FUNCTION_BLOCK FB_SaMElementUndefined EXTENDS FB_SaMElement
VAR
END_VAR

METHOD FB_init : BOOL
VAR_INPUT
	bInitRetains : BOOL; // if TRUE, the retain variables are initialized (warm start / cold start)
	bInCopyCode : BOOL;  // if TRUE, the instance afterwards gets moved into the copy code (online change)
END_VAR
THIS^.SetText (eLocation := E_BaseLocation.pl, wsDescription := "Nieokreślony");
THIS^.SetText (eLocation := E_BaseLocation.en, wsDescription := "Undefined");
THIS^.SetText (eLocation := E_BaseLocation.de, wsDescription := "Nicht definiert");
THIS^.SetName (stName := THIS^.GetTexts ());
END_METHOD

END_FUNCTION_BLOCK

(* stored: Version 1.1.0.1
   POU FB_SaMElementUndefined: Id {57cb239a-4f66-0563-155d-52bfe19a13e5}, SpecialFunc None
   Method FB_init: Id {8424b7bd-9912-08bf-2c92-b19073218c87} *)
